// TwinCAT 3 PLC project PLC
// ProgramVersion: 3.1.4026.14
// libraries:
//   Tc2_Standard, * (Beckhoff Automation GmbH)
//   Tc2_System, * (Beckhoff Automation GmbH)
//   Tc2_Utilities, * (Beckhoff Automation GmbH)
//   Tc3_EventLogger, * (Beckhoff Automation GmbH)
//   Tc3_Module, * (Beckhoff Automation GmbH)
// project tree:
//   Devices/ Machine_Info.TcDUT, Pelletizer.TcDUT, VFD.TcDUT
//   FBs/ F_DPLC.TcPOU, Hour_Meter_FB.TcPOU, Send_Event_FB.TcPOU, SlaveStatus_FB.TcPOU
//   Global_Machine/ GVL_AirKnife.TcGVL, GVL_Pelletizer.TcGVL, GVL_System.TcGVL, GVL_Waterbath.TcGVL
//   / PlcTask.TcTTO
//   POUs/AirKnife/ Air_Knife_Control_Word.TcPOU, Check_Filter.TcPOU
//   POUs/ Main.TcPOU
//   POUs/Pelletizer/ DPLC.TcPOU, Machine_Limits.TcPOU, Pelletizer_Control.TcPOU, Pellet_Calibration.TcPOU
//   POUs/System/ Events.TcPOU, Imperial_Metric_Switching.TcPOU, Machine_Status.TcPOU, Scaling_And_Conversions.TcPOU, WritePersistentData_POU.TcPOU
//   POUs/WaterBath/ WaterBath_Control.TcPOU, Waterbath_Temp_Control.TcPOU
// real-time tasks:
//   TASK PlcTask: cycle T#10ms, priority 6, ADS port 350
// I/O:
//   DEVICE Device 1 (EtherCAT), AmsNetId 10.0.1.72.2.1
//     Rotor Drive [i550 Cabinet V06.04.xx]
//     Feedroll Drive [i550 Cabinet V06.04.xx]
// variable links:
//   PLC/PLC Instance <-> Device 1 (EtherCAT)/Feedroll Drive
//     PlcTask Inputs/GVL_Pelletizer.MyPelletizer.Feedroll_VFD.VFD_Actual_Current <-> TPDO (A) user config/Actual current
//     PlcTask Inputs/GVL_Pelletizer.MyPelletizer.Feedroll_VFD.VFD_Actual_Speed <-> TPDO (A) Velocity/Actual speed
//     PlcTask Inputs/GVL_Pelletizer.MyPelletizer.Feedroll_VFD.VFD_Actual_Torque <-> TPDO (A) user config/Actual torque
//     PlcTask Inputs/GVL_Pelletizer.MyPelletizer.Feedroll_VFD.VFD_Connection_Status <-> InfoData/State
//     PlcTask Inputs/GVL_Pelletizer.MyPelletizer.Feedroll_VFD.VFD_DC_Bus_Voltage <-> TPDO (A) user config/DC-bus voltage
//     PlcTask Inputs/GVL_Pelletizer.MyPelletizer.Feedroll_VFD.VFD_Digital_Input_Status <-> TPDO (A) user config/Digital input status
//     PlcTask Inputs/GVL_Pelletizer.MyPelletizer.Feedroll_VFD.VFD_Status_Word <-> TPDO (A) Velocity/CiA status word
//     PlcTask Outputs/GVL_Pelletizer.MyPelletizer.Feedroll_VFD.VFD_Control_Word <-> RPDO (A) Velocity/CiA control word
//     PlcTask Outputs/GVL_Pelletizer.MyPelletizer.Feedroll_VFD.VFD_Set_Speed <-> RPDO (A) Velocity/Set speed
//   PLC/PLC Instance <-> Device 1 (EtherCAT)/Rotor Drive
//     PlcTask Inputs/GVL_Pelletizer.MyPelletizer.Rotor_VFD.VFD_Actual_Current <-> TPDO (A) user config/Actual current
//     PlcTask Inputs/GVL_Pelletizer.MyPelletizer.Rotor_VFD.VFD_Actual_Speed <-> TPDO (A) Velocity/Actual speed
//     PlcTask Inputs/GVL_Pelletizer.MyPelletizer.Rotor_VFD.VFD_Actual_Torque <-> TPDO (A) user config/Actual torque
//     PlcTask Inputs/GVL_Pelletizer.MyPelletizer.Rotor_VFD.VFD_Connection_Status <-> InfoData/State
//     PlcTask Inputs/GVL_Pelletizer.MyPelletizer.Rotor_VFD.VFD_DC_Bus_Voltage <-> TPDO (A) user config/DC-bus voltage
//     PlcTask Inputs/GVL_Pelletizer.MyPelletizer.Rotor_VFD.VFD_Digital_Input_Status <-> TPDO (A) user config/Digital input status
//     PlcTask Inputs/GVL_Pelletizer.MyPelletizer.Rotor_VFD.VFD_Status_Word <-> TPDO (A) Velocity/CiA status word
//     PlcTask Outputs/GVL_Pelletizer.MyPelletizer.Rotor_VFD.VFD_Control_Word <-> RPDO (A) Velocity/CiA control word
//     PlcTask Outputs/GVL_Pelletizer.MyPelletizer.Rotor_VFD.VFD_Set_Speed <-> RPDO (A) Velocity/Set speed

CONFIGURATION PLC
    RESOURCE PLC ON TwinCAT3
        TASK PlcTask(INTERVAL := T#10ms, PRIORITY := 6);
        PROGRAM Main WITH PlcTask : Main;
        PROGRAM Air_Knife_Control_Word WITH PlcTask : Air_Knife_Control_Word;
        PROGRAM Machine_Status WITH PlcTask : Machine_Status;
        PROGRAM WaterBath_Control WITH PlcTask : WaterBath_Control;
        PROGRAM Pelletizer_Control WITH PlcTask : Pelletizer_Control;
        PROGRAM Events WITH PlcTask : Events;
        PROGRAM WritePersistentData_POU WITH PlcTask : WritePersistentData_POU;
    END_RESOURCE
END_CONFIGURATION

// ---- Devices/Machine_Info.TcDUT
TYPE Machine_Info :
STRUCT
	Machine_Serial_Number : STRING;
	Electrical_Bill_ID : STRING;
	Purchase_Order_Number : STRING;
	Work_Order_Number : STRING;
END_STRUCT
END_TYPE

// ---- Devices/Pelletizer.TcDUT
TYPE Pelletizer :
STRUCT
	Feedroll_VFD : VFD;
	Rotor_VFD : VFD;

	
	Feedroll_Driven_Pulley : REAL := 1;
	Feedroll_Drive_Pulley : REAL := 1;
	Feedroll_Diameter_Inch : REAL := 1.88;
	Feedroll_RPM: INT;
	Feedroll_Motor_RPM : INT;
	Feedroll_Feet_Per_Minute : REAL;
	Feedroll_Meters_Per_Minute : REAL;

	
	Rotor_Driven_Pulley : REAL := 1;
	Rotor_Drive_Pulley : REAL := 1;
	Rotor_Tooth_Count : REAL := 32;
	Rotor_RPM_Limit : REAL:= 1000;
	Rotor_RPM : REAL;
	Rotor_Motor_RPM : REAL;


	Pellet_Length_Inch_Input : REAL := 0.125;
	Pellet_Length_Calibration_Value : REAL := 1;
	Pellet_Length_Measured_Input : REAL;			//For use in Calibration
	
	
	Pelletizer_Info : Machine_Info;
	
	Pelletizer_Start : BOOL;
	Pelletizer_Fault : BOOL;
	Pelletizer_Fault_Reset : BOOL;
	Pelletizer_STO : BOOL;
END_STRUCT
END_TYPE

// ---- Devices/VFD.TcDUT
TYPE VFD :		//Map these directly to the Process Data.
STRUCT
	// PLC Inputs (Data read from the inverter) TPDOs
	VFD_Status_Word AT %I* : UINT;												//CiA Status Word
	VFD_Actual_Speed AT %I* : INT;												//VFD Actual Output RPM 
	VFD_Error_Code AT %I* : UINT;												//Error Message
	VFD_Actual_Torque AT %I* : INT;												//Instantaneous Torque of the Motor (In Percent x.x%)
	VFD_Actual_Current AT %I* : UINT;											//Instantaneous Current of the Motor (In Percent x.x%)
	VFD_DC_Bus_Voltage AT %I* : UDINT;											//Instantaneous DC Bus Voltage of the VFD (x.xxx Volts)
	VFD_Digital_Input_Status AT %I* : UDINT;

	VFD_Fault : BOOL;		 //:= VFD_Status_Word.3;				This callout doesnt seem to work during Runtime.						//This is part of the Status Word; Fault bit 3
	VFD_Connection_Status AT %I* : UINT;
	

	// PLC Outputs (Data written to the inverter) RPDOs
	VFD_Control_Word AT %Q* : UINT;												//State Machine for Controlling VFD (CiA)
	VFD_Set_Speed AT %Q* : INT;													//Sets the Speed of the VFD in RPM
	VFD_DigitalOutput1_Word AT %Q* : UINT;										//Map the NetInWord2 to something we can use.

	VFD_DigitalOutput1_Bit : BOOL := VFD_DigitalOutput1_Word.0;					//Break out just the bit that we use to control the digital output
	VFD_Fault_Reset : BOOL;	// := VFD_Control_Word.7;				This callout doesnt seem to work during Runtime.				//This is part of the Control Word; Fault Reset bit 7
	
END_STRUCT
END_TYPE

// ---- Global_Machine/GVL_AirKnife.TcGVL
{attribute 'qualified_only'}
VAR_GLOBAL PERSISTENT
	AirKnife_VFD : VFD;
	AirKnife_Start : BOOL;
	AirKnife_Percent_Speed_Input : REAL := 100;
	AirKnife_StartwithSystem : BOOL;
	AirKnife_StopwithSystem : BOOL;
	AirKnife_Analog_Input AT %I* : INT;
	AirKnife_Filter_Change_Setting : REAL := 15;
	AirKnife_Vacuum_Level : REAL;
END_VAR

// ---- Global_Machine/GVL_Pelletizer.TcGVL
{attribute 'qualified_only'}
///PERSISTENT VARIABLES: retain their value after an uncontrolled termination, a Reset cold or a new download of the PLC project. 
VAR_GLOBAL PERSISTENT	
//MyPelletizer structure. This is the main reference to all major variables for a pelletizer. 
// To call variables throughout program: Ex) GVL_Pelletizer.MyPelletizer.Feedroll_Motor.Motor_Rated_RPM := 1755;
	MyPelletizer : Pelletizer;
////////////////////////////////////////////////////////////////////////////////////////////////////
	

	Pellet_Length_Incorrect : BOOL;
END_VAR

// ---- Global_Machine/GVL_System.TcGVL
{attribute 'qualified_only'}
VAR_GLOBAL PERSISTENT
	
	RunTime : REAL;
	Emergency_Stop_Active : BOOL;
	Metric_Set_Bit : BOOL;

END_VAR

// ---- Global_Machine/GVL_Waterbath.TcGVL
{attribute 'qualified_only'}
VAR_GLOBAL PERSISTENT
	//OUTPUTS
	Prop_Valve AT %Q* : INT; 
	Pump_Start AT %Q* : BOOL;
	Pump_OL_Reset AT %Q* : BOOL;

	//INPUTS
	Process_Water_IN AT %I* : INT;
	Process_Water_OUT AT %I* : INT;
	Process_Water_FLOW AT %I* : INT;
	Pellet_Temp_Probe AT %I* : INT;
	Process_Water_Setpoint : INT;
	Waterbath_Connection_Status AT %I* : UINT;
	Waterbath_System_Control AT %I* : BOOL;
	Pump_Fault AT %I* : BOOL;

	
	//System Variables
	Waterbath_StartwithSystem : BOOL;
	Waterbath_StopwithSystem : BOOL;
	Waterbath_Start : BOOL;
	Waterbath_Running : BOOL;
	Waterbath_Local_Control : BOOL;
	
	//These are the HMI Variables after they are scaled correctly.
	Waterbath_SetPoint_Temp : LREAL;
	Waterbath_Actual_Temp : LREAL;
	Waterbath_Return_Temp : REAL;
	Waterbath_Flow_Rate : REAL;
	Waterbath_Pellet_Temperature : REAL;
	
	Waterbath_TempControl_Auto : BOOL;

	Waterbath_Delta_Temp : REAL;
	Waterbath_CalculatedBTULoss : REAL;
	
	Waterbath_Valve_Position_Percentage : REAL;
	
END_VAR

// ---- POUs/Main.TcPOU
PROGRAM Main
VAR PERSISTENT

	Hour_Meter : Hour_Meter_FB;

	connected : BOOL;
END_VAR

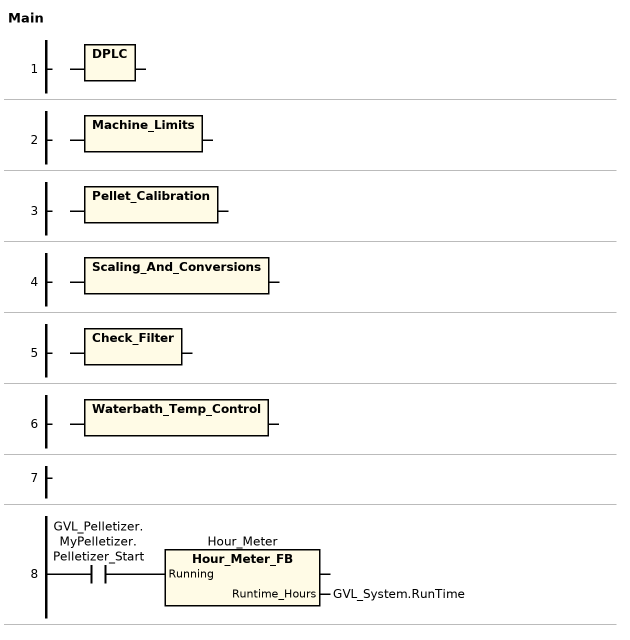
// NETWORK 1
DPLC();

// NETWORK 2
Machine_Limits();

// NETWORK 3
Pellet_Calibration();

// NETWORK 4
Scaling_And_Conversions();

// NETWORK 5
Check_Filter();

// NETWORK 6
Waterbath_Temp_Control();

// NETWORK 7

// NETWORK 8
Hour_Meter(Running := GVL_Pelletizer.MyPelletizer.Pelletizer_Start, Runtime_Hours => GVL_System.RunTime); // Hour_Meter_FB

END_PROGRAM

// ---- FBs/Hour_Meter_FB.TcPOU
FUNCTION_BLOCK Hour_Meter_FB
VAR_INPUT
	Running : BOOL;
END_VAR
VAR_OUTPUT
	Runtime_Hours : REAL;
END_VAR
VAR
	Running_Temp : BOOL;
	Minute_Timer : TON;
	Minutes : REAL;
	Hours : REAL;
	Elapsed : TIME;
END_VAR

Minute_Timer(IN:=Running_Temp , PT:=T#60S , Q=>, ET=>Elapsed );

IF Running THEN
	Running_Temp := TRUE;
END_IF
IF Minute_Timer.Q THEN
	Running_Temp := FALSE;
	Minutes := Minutes + 1;
END_IF
IF Minutes >= 60 THEN
	Minutes := 0;
	Hours := Hours + 1;
END_IF

Runtime_Hours := Hours;

END_FUNCTION_BLOCK

// ---- POUs/Pelletizer/DPLC.TcPOU
PROGRAM DPLC
VAR
	DPLC : F_DPLC;

	Calibrated_Pellet_Length : REAL;
END_VAR

GVL_Pelletizer.MyPelletizer.Feedroll_Motor_RPM := GVL_Pelletizer.MyPelletizer.Feedroll_VFD.VFD_Actual_Speed;

Calibrated_Pellet_Length := GVL_Pelletizer.MyPelletizer.Pellet_Length_Inch_Input * GVL_Pelletizer.MyPelletizer.Pellet_Length_Calibration_Value;

DPLC(
	Pellet_Length_Inch_Input		:= Calibrated_Pellet_Length,
	Feedroll_Diameter				:= GVL_Pelletizer.MyPelletizer.Feedroll_Diameter_Inch,
	Feedroll_Drive_Gear				:= GVL_Pelletizer.MyPelletizer.Feedroll_Drive_Pulley,
	Feedroll_Driven_Gear			:= GVL_Pelletizer.MyPelletizer.Feedroll_Driven_Pulley,
	Feedroll_Motor_RPM				:= GVL_Pelletizer.MyPelletizer.Feedroll_Motor_RPM,
	Rotor_Drive_Gear				:= GVL_Pelletizer.MyPelletizer.Rotor_Drive_Pulley,
	Rotor_Driven_Gear				:= GVL_Pelletizer.MyPelletizer.Rotor_Driven_Pulley,
	Rotor_Tooth_Count				:= GVL_Pelletizer.MyPelletizer.Rotor_Tooth_Count,
	Rotor_Motor_RPM					=> GVL_Pelletizer.MyPelletizer.Rotor_Motor_RPM,
	Rotor_RPM						=> GVL_Pelletizer.MyPelletizer.Rotor_RPM,
	Feedroll_Feet_Per_Minute		=> GVL_Pelletizer.MyPelletizer.Feedroll_Feet_Per_Minute
);
	
GVL_Pelletizer.MyPelletizer.Rotor_VFD.VFD_Set_Speed := REAL_TO_INT(GVL_Pelletizer.MyPelletizer.Rotor_Motor_RPM);


//Check for rotor speed exceeded. 
IF GVL_Pelletizer.MyPelletizer.Rotor_RPM >= GVL_Pelletizer.MyPelletizer.Rotor_RPM_Limit THEN
	GVL_Pelletizer.Pellet_Length_Incorrect := TRUE;
ELSE	
	GVL_Pelletizer.Pellet_Length_Incorrect := FALSE;
END_IF

END_PROGRAM

// ---- FBs/F_DPLC.TcPOU
FUNCTION_BLOCK F_DPLC
VAR_INPUT
	Pellet_Length_Inch_Input : REAL;
	
	//Feedroll
	Feedroll_Diameter : REAL;
	Feedroll_Drive_Gear : REAL;
	Feedroll_Driven_Gear : REAL;
	Feedroll_Motor_RPM : REAL;
	
	//Rotor
	Rotor_Drive_Gear : REAL;
	Rotor_Driven_Gear : REAL;
	Rotor_Tooth_Count : REAL;
	
END_VAR
VAR_OUTPUT
	
	Rotor_Motor_RPM : REAL;	//Commands the motor speed
	Rotor_RPM : REAL;		//Displays the actualy Rotor Speed
	
	Feedroll_Feet_Per_Minute : REAL;	//Displays the Actual Ft/min

END_VAR
VAR
	Feedroll_RPM : REAL;
	Feedroll_Inch_Per_Minute : REAL;

	Rotor_Cuts_Per_Minute : REAL;
END_VAR

Feedroll_RPM := Feedroll_Motor_RPM * (Feedroll_Drive_Gear / Feedroll_Driven_Gear);

Feedroll_Inch_Per_Minute := Feedroll_RPM * (Feedroll_Diameter * 3.14159);

Feedroll_Feet_Per_Minute := Feedroll_Inch_Per_Minute / 12.0;




Rotor_Cuts_Per_Minute := Feedroll_Inch_Per_Minute / Pellet_Length_Inch_Input;

Rotor_RPM := Rotor_Cuts_Per_Minute / Rotor_Tooth_Count;

Rotor_Motor_RPM := Rotor_RPM / (Rotor_Drive_Gear / Rotor_Driven_Gear);

END_FUNCTION_BLOCK

// ---- POUs/Pelletizer/Machine_Limits.TcPOU
PROGRAM Machine_Limits
VAR PERSISTENT
//For calculation purposes only. This calculates the min and max line speeds so that we can display these ranges on the speed gauges.

Feedroll_Motor_Rated_RPM : REAL := 1750;	
Feedroll_Motor_Rated_Hz : REAL := 60;		
Feedroll_Motor_Maximum_Hz : REAL;	
Feedroll_Motor_Minimum_Hz : REAL;	
Feedroll_Max_Ft_Per_Min : REAL;
Feedroll_Min_Ft_Per_Min  : REAL;
Feedroll_Motor_RPM_Per_Hz : REAL;
Feedroll_Pulley_Ratio : REAL;
Feedroll_Circumference_Feet : REAL := (GVL_Pelletizer.MyPelletizer.Feedroll_Diameter_Inch * 3.14159) / 12.0;

Rotor_Motor_Rated_RPM : REAL := 1750;	
Rotor_Motor_Rated_Hz : REAL := 60;	
Rotor_Motor_Maximum_Hz : REAL;	
Rotor_Motor_Minimum_Hz : REAL;	
Rotor_Max_RPM : REAL;
Rotor_Min_RPM : REAL;
Rotor_Motor_RPM_Per_Hz : REAL;
Rotor_Pulley_Ratio : REAL;


END_VAR

Feedroll_Pulley_Ratio := (GVL_Pelletizer.MyPelletizer.Feedroll_Drive_Pulley / GVL_Pelletizer.MyPelletizer.Feedroll_Driven_Pulley);

Feedroll_Motor_RPM_Per_Hz := Feedroll_Motor_Rated_RPM / Feedroll_Motor_Rated_Hz;

Feedroll_Max_Ft_Per_Min := ((Feedroll_Motor_RPM_Per_Hz * Feedroll_Motor_Maximum_Hz) * Feedroll_Pulley_Ratio) * Feedroll_Circumference_Feet;

Feedroll_Min_Ft_Per_Min := ((Feedroll_Motor_RPM_Per_Hz * Feedroll_Motor_Minimum_Hz) * Feedroll_Pulley_Ratio) * Feedroll_Circumference_Feet;



Rotor_Pulley_Ratio := (GVL_Pelletizer.MyPelletizer.Rotor_Drive_Pulley / GVL_Pelletizer.MyPelletizer.Rotor_Driven_Pulley);

Rotor_Motor_RPM_Per_Hz := Rotor_Motor_Rated_RPM / Rotor_Motor_Rated_Hz;

Rotor_Max_RPM := (Rotor_Motor_RPM_Per_Hz * Rotor_Motor_Maximum_Hz) * Rotor_Pulley_Ratio;

Rotor_Min_RPM := (Rotor_Motor_RPM_Per_Hz * Rotor_Motor_Minimum_Hz) * Rotor_Pulley_Ratio;

END_PROGRAM

// ---- POUs/Pelletizer/Pellet_Calibration.TcPOU
PROGRAM Pellet_Calibration
VAR
	SET_CALIBRATON_VALUE : BOOL;

	
	
	Pellet_Length_Temp_Cal_Val : REAL;
END_VAR

 Pellet_Length_Temp_Cal_Val :=  GVL_Pelletizer.MyPelletizer.Pellet_Length_Inch_Input / GVL_Pelletizer.MyPelletizer.Pellet_Length_Measured_Input;


IF SET_CALIBRATON_VALUE THEN
	GVL_Pelletizer.MyPelletizer.Pellet_Length_Calibration_Value := Pellet_Length_Temp_Cal_Val;
END_IF

END_PROGRAM

// ---- POUs/System/Scaling_And_Conversions.TcPOU
PROGRAM Scaling_And_Conversions
VAR
	Rotor_Actual_Torque_Scaled : REAL;
	Feedroll_Actual_Torque_Scaled : REAL;
	
	Rotor_Actual_Current_Scaled : REAL;
	Feedroll_Actual_Current_Scaled : REAL;
	AirKnife_Actual_Current_Scaled : REAL;
	
	Rotor_DC_Bus_Voltage_Scaled : REAL;
	Feedroll_DC_Bus_Voltage_Scaled : REAL;
	AirKnife_DC_Bus_Voltage_Scaled : REAL;
	

	AirKnife_Vacuum_Scaler : REAL := -4.0176; //-401.76 inH2O (-14.5PSI) / 100% = 4.0176
	
END_VAR

Rotor_Actual_Torque_Scaled := INT_TO_REAL(GVL_Pelletizer.MyPelletizer.Rotor_VFD.VFD_Actual_Torque) / 10;
Feedroll_Actual_Torque_Scaled := INT_TO_REAL(GVL_Pelletizer.MyPelletizer.Feedroll_VFD.VFD_Actual_Torque) / 10;

Rotor_Actual_Current_Scaled := UINT_TO_REAL(GVL_Pelletizer.MyPelletizer.Rotor_VFD.VFD_Actual_Current) / 10;
Feedroll_Actual_Current_Scaled := UINT_TO_REAL(GVL_Pelletizer.MyPelletizer.Feedroll_VFD.VFD_Actual_Current) / 10;
AirKnife_Actual_Current_Scaled := UINT_TO_REAL(GVL_Airknife.AirKnife_VFD.VFD_Actual_Current) / 10;


Rotor_DC_Bus_Voltage_Scaled := UDINT_TO_REAL(GVL_Pelletizer.MyPelletizer.Rotor_VFD.VFD_DC_Bus_Voltage) / 1000;
Feedroll_DC_Bus_Voltage_Scaled := UDINT_TO_REAL(GVL_Pelletizer.MyPelletizer.Feedroll_VFD.VFD_DC_Bus_Voltage) / 1000;
AirKnife_DC_Bus_Voltage_Scaled := UDINT_TO_REAL(GVL_AirKnife.AirKnife_Vfd.VFD_DC_Bus_Voltage) / 1000;

GVL_Airknife.AirKnife_Vacuum_Level := INT_TO_REAL(GVL_AirKnife.AirKnife_Analog_Input / 10) * AirKnife_Vacuum_Scaler;
//Sensor Scale:
//100% = -401.76 Inches of Water
//0% = 0 inches of water
//The analog input is read in as a percentage, not as 4-20ma

GVL_Waterbath.Waterbath_Actual_Temp := (((INT_TO_REAL(GVL_Waterbath.Process_Water_OUT) / 10) * 1.8) + 32.0);	//Convert thermocouple to Degrees F. 
GVL_Waterbath.Waterbath_Return_Temp := ((INT_TO_REAL(GVL_Waterbath.Process_Water_IN) / 30518.0) * 158);	//14F Degrees = 0 ADC; //158F Degrees = 30518
GVL_Waterbath.Waterbath_Pellet_Temperature := (((INT_TO_REAL(GVL_Waterbath.Pellet_Temp_Probe) / 10) * 1.8) + 32.0); //Convert thermocouple to Degrees F.

//0 - 198.129 GPM
GVL_Waterbath.Waterbath_Flow_Rate := ((INT_TO_REAL(GVL_WAterbath.Process_Water_FLOW) / 30518.0) * 198.129);

END_PROGRAM

// ---- POUs/AirKnife/Check_Filter.TcPOU
PROGRAM Check_Filter
VAR
	Change_Filter : BOOL;
	Startup_Timer : TON;
END_VAR

Startup_Timer(IN := GVL_airknife.AirKnife_Start,PT:=T#15S);	//Dont flag an alarm while it is starting up. Give it 15 seconds


IF (GVL_AirKnife.AirKnife_Filter_Change_Setting <= GVL_AirKnife.AirKnife_Vacuum_Level) AND (GVL_AirKnife.AirKnife_Vacuum_Level < -0.2) AND Startup_Timer.Q THEN
	Change_Filter := TRUE;
ELSE
	Change_Filter := FALSE;
END_IF

END_PROGRAM

// ---- POUs/WaterBath/Waterbath_Temp_Control.TcPOU
PROGRAM Waterbath_Temp_Control
VAR PERSISTENT
	Cooling_PID: FB_BasicPID;
	
	WaterbathPID_CycleTime : LREAL;
	Waterbath_ResetPID : BOOL;
	WaterbathPID_Kp : LREAL;
	WaterbathPID_Tn : LREAL;
	WaterbathPID_Tv : LREAL;
	WaterbathPID_Td : LREAL;
	
	WaterbathPID_ControlOutput : LREAL;
	WaterbathPID_ControlOutput_Temp : LREAL;

	WaterbathPID_ErrorStatus : UINT;
	
	
	
	
	//Erics Proportional Control
	
	Error : REAL;
	Gain : REAL;
	Deadband : REAL;
	
END_VAR

IF GVL_Waterbath.Waterbath_TempControl_Auto THEN
//	Cooling_PID(
//	fSetpointValue:= GVL_Waterbath.Waterbath_SetPoint_Temp, 
//	fActualValue:= GVL_Waterbath.Waterbath_Actual_Temp, 
//	bReset:= Waterbath_ResetPID, 
//	fCtrlCycleTime:= WaterbathPID_CycleTime, 
//	fKp:= WaterbathPID_Kp, 
//	fTn:= WaterbathPID_Tn, 
//	fTv:= WaterbathPID_Tv, 
//	fTd:= WaterbathPID_Td, 
//	fCtrlOutput=> WaterbathPID_ControlOutput, 
//	nErrorStatus=> WaterbathPID_ErrorStatus);


//Erics Proportional Algorithm
//Calculate error in temp difference
	Error := (GVL_Waterbath.Waterbath_Actual_Temp - GVL_Waterbath.Waterbath_SetPoint_Temp);	
//See if error is within deadband of 2 degrees
	IF ABS(Error) < Deadband THEN
		Error := 0;
	END_IF
//Error times the gain to set the output
	WaterbathPID_ControlOutput_Temp := Error * Gain;
//Limits on output. 	
	IF WaterbathPID_ControlOutput_Temp >= 100 THEN
		WaterbathPID_ControlOutput_Temp := 100;
	ELSIF WaterbathPID_ControlOutput_Temp < 0 THEN
		WaterbathPID_ControlOutput_Temp := 0;
	END_IF
	
	GVL_Waterbath.Waterbath_Valve_Position_Percentage := WaterbathPID_ControlOutput_Temp;
	WaterbathPID_ControlOutput := (GVL_Waterbath.Waterbath_Valve_Position_Percentage / 100) * 30518.0;
ELSE
	WaterbathPID_ControlOutput := (GVL_Waterbath.Waterbath_Valve_Position_Percentage / 100) * 30518.0;
END_IF

GVL_Waterbath.Prop_Valve := LREAL_TO_INT(WaterbathPID_ControlOutput);



GVL_Waterbath.Waterbath_Delta_Temp := GVL_Waterbath.Waterbath_Return_Temp - GVL_Waterbath.Waterbath_Actual_Temp;
GVL_Waterbath.Waterbath_CalculatedBTULoss := (GVL_Waterbath.Waterbath_Flow_Rate * (GVL_Waterbath.Waterbath_Delta_Temp) * 500.4);
// BTU Loss = Flow Rate In GPM (of water) x (Temperature Leaving Process - Temperature Entering Process) x 500.4

END_PROGRAM

// ---- POUs/AirKnife/Air_Knife_Control_Word.TcPOU
PROGRAM Air_Knife_Control_Word
VAR
	
	AirKnife_Lower_Status_Byte : UINT;
	
	Status_BitMask : UINT := 65280;

	
	Estop_Temp : bool;
END_VAR

GVL_AirKnife.AirKnife_VFD.VFD_Fault := GVL_AirKnife.AirKnife_VFD.VFD_Status_Word.3;	//Set fault bit equal to the status word fault bit.

IF GVL_AirKnife.AirKnife_VFD.VFD_Fault_Reset THEN
	//if the fault reset button was pressed, set the fault reset bit in the control word.
	GVL_AirKnife.AirKnife_VFD.VFD_Control_Word.7 := TRUE;
ELSE
	GVL_AirKnife.AirKnife_VFD.VFD_Control_Word.7 := FALSE;
END_IF



IF GVL_AirKnife.AirKnife_VFD.VFD_Fault THEN
	//If Faulted, then switch off drives
	GVL_AirKnife.AirKnife_VFD.VFD_Control_Word.0 := FALSE;
END_IF



IF GVL_Airknife.AirKnife_Stopwithsystem THEN
	Estop_Temp := GVL_Pelletizer.MyPelletizer.Pelletizer_STO;
ELSE
	Estop_Temp := TRUE;
END_IF

IF GVL_AirKnife.AirKnife_StartwithSystem THEN
	GVL_Airknife.AirKnife_Start := GVL_Pelletizer.MyPelletizer.Pelletizer_Start;
END_IF


	//If the Start button on the HMI is pressed, OR it is set to start with the rest of the system. The checkbox must be set and pelletizer must be started.
IF GVL_AirKnife.AirKnife_Start AND Estop_Temp THEN
	
//Feedroll Case Statement
	AirKnife_Lower_Status_Byte := GVL_AirKnife.AirKnife_VFD.VFD_Status_Word OR Status_BitMask;	// Bitwise OR with bits 7-15 of status word because we dont care about them for control.
	
	CASE AirKnife_Lower_Status_Byte OF
		65392: //Voltage Enabled, Switch On Disabled.
		GVL_AirKnife.AirKnife_VFD.VFD_Control_Word := 6;	//Enable Voltage, Disable Quick Stop	
	
		65360: //Voltage Enabled, Switch On Disabled.
		GVL_AirKnife.AirKnife_VFD.VFD_Control_Word := 6;	//Enable Voltage, Disable Quick Stop
	
		65329: //Ready To Switch On, Voltage Enabled, Quick Stop Disabled.
		GVL_AirKnife.AirKnife_VFD.VFD_Control_Word := 7;	//Enable Voltage, Disable Quick Stop, Switch On
	
		65331: //Ready To Switch On, Switched On, Voltage Enabled, Quick Stop Disabled.
		GVL_AirKnife.AirKnife_VFD.VFD_Control_Word := 15;	//Enable Voltage, Disable Quick Stop, Switch On, Enable Operation
	
		65335: //Ready To Switch On, Switched On, Operation Enabled, Voltage Enabled, Quick Stop Disabled.
		GVL_AirKnife.AirKnife_VFD.VFD_Control_Word.0 := TRUE;	//Switch On Bit. 
	END_CASE;

ELSE	
	//If we are not running, switch off Drives
	GVL_AirKnife.AirKnife_VFD.VFD_Control_Word.0 := 0;
END_IF



//The last thing is to scale the motor RPM to a percentage.
GVL_AirKnife.AirKnife_VFD.VFD_Set_Speed := REAL_TO_INT((3450 / 100) * GVL_AirKnife.AirKnife_Percent_Speed_Input);
// I should add some parameters for the air knife settings screen to the max RPM

END_PROGRAM

// ---- POUs/System/Machine_Status.TcPOU
PROGRAM Machine_Status
VAR
	AirKnife_Status_String : STRING;
	AirKnife_Disconnected : BOOL;
	AirKnife_Connected : bool;
	
	Rotor_Status_String : STRING;
	Rotor_Disconnected : BOOL;
	
	Feedroll_Status_String : STRING;
	Feedroll_Disconnected : BOOL;
	
	Pelletizer_Status_String : STRING;
	
	Waterbath_Status_String : STRING;
	Waterbath_Disconnected : BOOL;
	Waterbath_Connected : BOOL;
	
END_VAR


Rotor_Status_String := SlaveStatus_FB(GVL_Pelletizer.MyPelletizer.Rotor_VFD.VFD_Connection_Status, Slave_Disconnected => Rotor_Disconnected);
Feedroll_Status_String := SlaveStatus_FB(GVL_Pelletizer.MyPelletizer.Feedroll_VFD.VFD_Connection_Status, Slave_Disconnected => Feedroll_Disconnected);

IF Rotor_Disconnected OR Feedroll_Disconnected THEN
	Pelletizer_Status_String := CONCAT(Rotor_Status_String, Feedroll_Status_String);
ELSE
	Pelletizer_Status_String := 'Slave in OP state';
END_IF


AirKnife_Status_String := SlaveStatus_FB(GVL_AirKnife.AirKnife_VFD.VFD_Connection_Status, Slave_Disconnected => AirKnife_Disconnected);
AirKnife_connected := NOT Airknife_Disconnected;

Waterbath_Status_String := SlaveStatus_FB(GVL_Waterbath.Waterbath_Connection_Status, Slave_Disconnected => Waterbath_Disconnected);
Waterbath_Connected := NOT Waterbath_Disconnected;

END_PROGRAM

// ---- FBs/SlaveStatus_FB.TcPOU
FUNCTION SlaveStatus_FB : STRING
VAR_INPUT
	InfoData_State : UINT; // Input variable containing the status bitmask
END_VAR
VAR
	Bit8_Message : STRING;
	Bitmask : UINT := 16#FFF0;
	Masked_State: UINT;
END_VAR
VAR_OUTPUT
	Slave_Disconnected : BOOL;
END_VAR

Masked_State := bitmask OR InfoData_State;


IF InfoData_State.8 THEN
	Bit8_Message := ' - Slave NOT present ';
	Slave_Disconnected := TRUE;
ELSE
	Bit8_Message := '';
	Slave_Disconnected := FALSE;
END_IF
	



CASE Masked_State OF
    16#FFF1: SlaveStatus_FB 		:= 'Slave in INIT state';		//16#___1; // Slave in 'INIT' state
    16#FFF2: SlaveStatus_FB 		:= 'Slave in PREOP state';		//16#___2; // Slave in 'PREOP' state
    16#FFF3: SlaveStatus_FB 		:= 'Slave in BOOT state';		//16#___3; // Slave in 'BOOT' state
    16#FFF4: SlaveStatus_FB 		:= 'Slave in SAFEOP state';		//16#___4; // Slave in 'SAFEOP' state
    16#FFF8: SlaveStatus_FB 		:= 'Slave in OP state';			//16#___8 Slave in 'OP' state
ELSE
    // Handle invalid input or unknown status
    SlaveStatus_FB := 'Abnormal Status'; // Set an appropriate error value
	Slave_Disconnected := TRUE;
END_CASE;

SlaveStatus_FB := CONCAT(SlaveStatus_FB, Bit8_message);	//Add both messages to display.



//Breakdown of Statuses for Infomation, we dont care about all of them. Just the EtherCAT State and the slave Not present bit. 
//0x___1 = Slave in 'INIT' state
//0x___2 = Slave in 'PREOP' state
//0x___3 = Slave in 'BOOT' state
//0x___4 = Slave in 'SAFEOP' state
//0x___8 = Slave in 'OP' state
//0x001_ = Slave signals error
//0x002_ = Invalid vendorId, productCode... read
//0x004_ = Initialization error occurred
//0x008_ = Slave disabled
//0x010_ = Slave not present
//0x020_ = Slave signals link error
//0x040_ = Slave signals missing link
//0x080_ = Slave signals unexpected link
//0x100_ = Communication port A
//0x200_ = Communication port B
//0x400_ = Communication port C
//0x800_ = Communication port D

END_FUNCTION

// ---- POUs/WaterBath/WaterBath_Control.TcPOU
PROGRAM WaterBath_Control
VAR
	
	Estop_Temp : bool;

END_VAR

IF GVL_Waterbath.Waterbath_StopwithSystem THEN		//if the pelletizer estop is pressed AND the setting for system stop is set, then stop with an estop.
	Estop_Temp := GVL_Pelletizer.MyPelletizer.Pelletizer_STO;
ELSE
	Estop_Temp := TRUE;
END_IF




IF GVL_Waterbath.Waterbath_StartwithSystem THEN
	GVL_Waterbath.Waterbath_Start := GVL_Pelletizer.MyPelletizer.Pelletizer_Start;
END_IF




IF GVL_Waterbath.Waterbath_Start AND Estop_Temp THEN
	GVL_Waterbath.Pump_Start := TRUE;
ELSE
	GVL_Waterbath.Pump_Start := FALSE;
END_IF


GVL_Waterbath.Waterbath_Local_Control := NOT GVL_Waterbath.Waterbath_System_Control;

END_PROGRAM

// ---- POUs/Pelletizer/Pelletizer_Control.TcPOU
PROGRAM Pelletizer_Control
VAR
	Pelletizer_Lower_Status_Byte : UINT;
	
	Status_BitMask : UINT := 65280;
	DigitalInputStatus: INT;
	


END_VAR

//Bit 15 is digital input 1 which is the pelletizer control relay. If both of these are ON, we are in a started state.
IF (GVL_Pelletizer.MyPelletizer.Feedroll_VFD.VFD_Digital_Input_Status.16 = TRUE) AND (GVL_Pelletizer.MyPelletizer.Rotor_VFD.VFD_Digital_Input_Status.16 = TRUE) THEN
	GVL_Pelletizer.MyPelletizer.Pelletizer_Start := TRUE;
ELSE	
	GVL_Pelletizer.MyPelletizer.Pelletizer_Start := FALSE;
END_IF




//Fault Handling
GVL_Pelletizer.MyPelletizer.Feedroll_VFD.VFD_Fault := GVL_Pelletizer.MyPelletizer.Feedroll_VFD.VFD_Status_Word.3;
GVL_Pelletizer.MyPelletizer.Rotor_VFD.VFD_Fault := GVL_Pelletizer.MyPelletizer.Rotor_VFD.VFD_Status_Word.3;
//Overall Machine Fault if one or both drives faulted. 
IF (GVL_Pelletizer.MyPelletizer.Feedroll_VFD.VFD_Fault) OR (GVL_Pelletizer.MyPelletizer.Rotor_VFD.VFD_Fault) THEN
	GVL_Pelletizer.MyPelletizer.Pelletizer_Fault := TRUE;
ELSE
	GVL_Pelletizer.MyPelletizer.Pelletizer_Fault := FALSE;	
END_IF



//Reset faults
IF GVL_Pelletizer.MyPelletizer.Pelletizer_Fault_Reset THEN
	GVL_Pelletizer.MyPelletizer.Feedroll_VFD.VFD_Fault_Reset := TRUE;
	GVL_Pelletizer.MyPelletizer.Rotor_VFD.VFD_Fault_Reset := TRUE;
ELSE
	GVL_Pelletizer.MyPelletizer.Feedroll_VFD.VFD_Fault_Reset := FALSE;
	GVL_Pelletizer.MyPelletizer.Rotor_VFD.VFD_Fault_Reset := FALSE;
END_IF
//Set Reset
GVL_Pelletizer.MyPelletizer.Feedroll_VFD.VFD_Control_Word.7 := GVL_Pelletizer.MyPelletizer.Feedroll_VFD.VFD_Fault_reset;
GVL_Pelletizer.MyPelletizer.Rotor_VFD.VFD_Control_Word.7 := GVL_Pelletizer.MyPelletizer.Rotor_VFD.VFD_Fault_Reset;

GVL_Pelletizer.MyPelletizer.Pelletizer_STO := GVL_Pelletizer.MyPelletizer.Feedroll_VFD.VFD_Status_Word.15 OR GVL_Pelletizer.MyPelletizer.rotor_VFD.VFD_Status_Word.15;

END_PROGRAM

// ---- POUs/System/Events.TcPOU
PROGRAM Events
VAR
	Send_Start_Event : Send_Event_FB;
	Start_Event  : TcEventEntry := TC_Events.Pelletizer_Events.Start_Button_Event;
	
	Send_Stop_Event : Send_Event_FB;
	Stop_Event  : TcEventEntry := TC_Events.Pelletizer_Events.Stop_Button_Event;
//////////////////////////////////////////////////////////////////////////////////////////////////////////////////
	Send_EmergencyStop_Event : Send_Event_FB;
	EmergencyStop_Event : TcEventEntry := TC_Events.Pelletizer_Events.Emergency_Stop_Set_Event;

	Send_EmergencyStop_Reset_Event : Send_Event_FB;
	EmergencyStop_Reset_Event : TcEventEntry := TC_Events.Pelletizer_Events.Emergency_Stop_Reset_Event;
//////////////////////////////////////////////////////////////////////////////////////////////////////////////////	
	Send_Feedroll_Drive_Fault_Event : Send_Event_FB;
	Feedroll_Drive_Fault_Event : TcEventEntry := TC_Events.Pelletizer_Events.Feedroll_Drive_Fault_Event;
	
	Send_Feedroll_Drive_Fault_Reset_Event : Send_Event_FB;
	Feedroll_Drive_Fault_Reset_Event : TcEventEntry := TC_Events.Pelletizer_Events.Feedroll_Drive_Fault_Reset_Event;
//////////////////////////////////////////////////////////////////////////////////////////////////////////////////	
	Send_Rotor_Drive_Fault_Event : Send_Event_FB;
	Rotor_Drive_Fault_Event : TcEventEntry := TC_Events.Pelletizer_Events.Rotor_Drive_Fault_Event;
	
	Send_Rotor_Drive_Fault_Reset_Event : Send_Event_FB;
	Rotor_Drive_Fault_Reset_Event : TcEventEntry := TC_Events.Pelletizer_Events.Rotor_Drive_Fault_Reset_Event;
//////////////////////////////////////////////////////////////////////////////////////////////////////////////////
	Send_Machine_Shutdown_Event : Send_Event_FB;
	Machine_Shutdown_Event : TcEventEntry := TC_Events.Pelletizer_Events.Machine_Shutdown_Event;	
	
	Send_Machine_PowerOn_Event : Send_Event_FB;
	Machine_PowerOn_Event : TcEventEntry := TC_Events.Pelletizer_Events.Machine_PowerOn_Event;
//////////////////////////////////////////////////////////////////////////////////////////////////////////////////	
	Send_Exceeded_Pellet_Length_Event : Send_Event_FB;
	Exceeded_Pellet_Length_Event : TcEventEntry := TC_Events.Pelletizer_Events.PelletLength_Exceeded_Event;	
//////////////////////////////////////////////////////////////////////////////////////////////////////////////////	
	Send_Change_Filter_Event : Send_Event_FB;
	Change_Filter_Event : TcEventEntry := TC_Events.AirKnife_Events.Change_Filter_Event;	
	
	Send_Filter_OKAY_Event : Send_Event_FB;
	Filter_OKAY_Event : TcEventEntry := TC_Events.AirKnife_Events.Filter_OKAY_Event;
//////////////////////////////////////////////////////////////////////////////////////////////////////////////////	
	Send_Local_Mode_Active : Send_Event_FB;
	Local_Mode_Active : TcEventEntry := TC_Events.Waterbath_Events.Local_Mode_Active;
	
	Send_Remote_Mode_Active : Send_Event_FB;
	Remote_Mode_Active : TcEventEntry := TC_Events.Waterbath_Events.Remote_Mode_Active;
//////////////////////////////////////////////////////////////////////////////////////////////////////////////////	
	Send_Pump_Start_Event : Send_Event_FB;
	Pump_Start_Event : TcEventEntry := TC_Events.Waterbath_Events.Pump_Start_Event;
	
	Send_Pump_Stop_Event : Send_Event_FB;
	Pump_Stop_Event : TcEventEntry := TC_Events.Waterbath_Events.Pump_Stop_Event;
//////////////////////////////////////////////////////////////////////////////////////////////////////////////////	
	
	First_Scan : BOOL := False;	
END_VAR

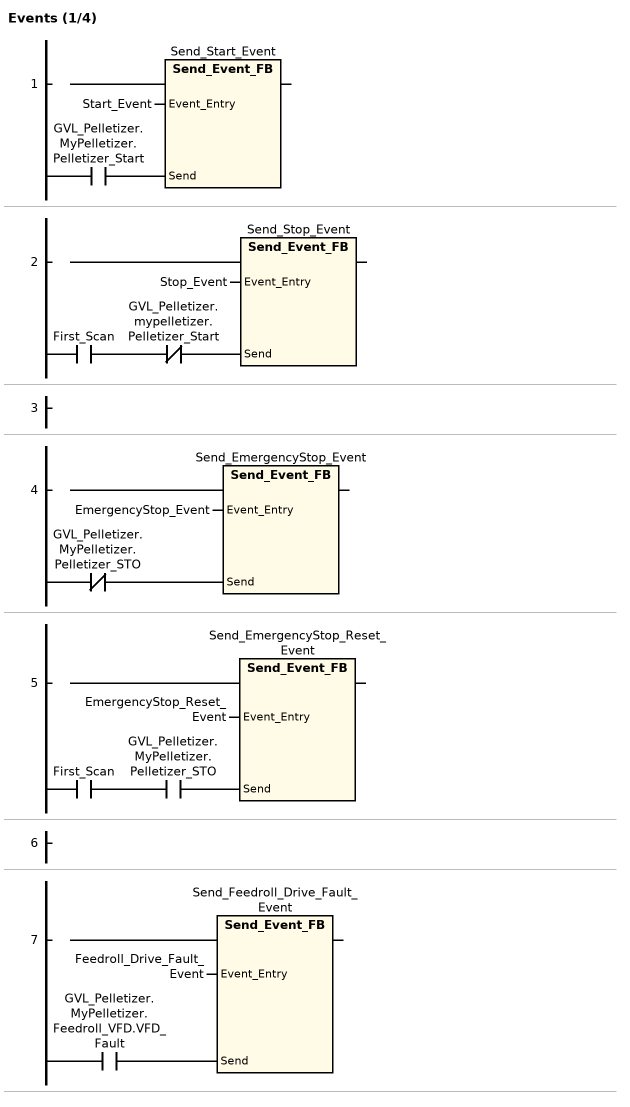
// NETWORK 1
Send_Start_Event(Event_Entry := Start_Event, Send := GVL_Pelletizer.MyPelletizer.Pelletizer_Start); // Send_Event_FB

// NETWORK 2
Send_Stop_Event(Event_Entry := Stop_Event, Send := First_Scan AND NOT GVL_Pelletizer.mypelletizer.Pelletizer_Start); // Send_Event_FB

// NETWORK 3

// NETWORK 4
Send_EmergencyStop_Event(Event_Entry := EmergencyStop_Event, Send := NOT GVL_Pelletizer.MyPelletizer.Pelletizer_STO); // Send_Event_FB

// NETWORK 5
Send_EmergencyStop_Reset_Event(Event_Entry := EmergencyStop_Reset_Event, Send := First_Scan AND GVL_Pelletizer.MyPelletizer.Pelletizer_STO); // Send_Event_FB

// NETWORK 6

// NETWORK 7
Send_Feedroll_Drive_Fault_Event(Event_Entry := Feedroll_Drive_Fault_Event, Send := GVL_Pelletizer.MyPelletizer.Feedroll_VFD.VFD_Fault); // Send_Event_FB

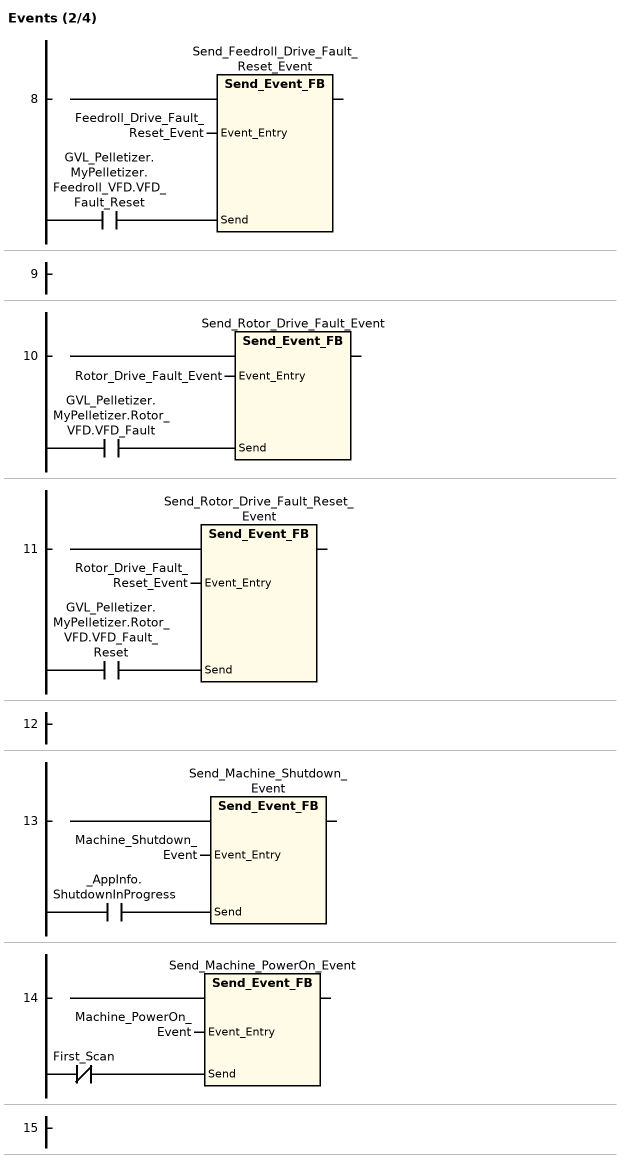
// NETWORK 8
Send_Feedroll_Drive_Fault_Reset_Event(Event_Entry := Feedroll_Drive_Fault_Reset_Event, Send := GVL_Pelletizer.MyPelletizer.Feedroll_VFD.VFD_Fault_Reset); // Send_Event_FB

// NETWORK 9

// NETWORK 10
Send_Rotor_Drive_Fault_Event(Event_Entry := Rotor_Drive_Fault_Event, Send := GVL_Pelletizer.MyPelletizer.Rotor_VFD.VFD_Fault); // Send_Event_FB

// NETWORK 11
Send_Rotor_Drive_Fault_Reset_Event(Event_Entry := Rotor_Drive_Fault_Reset_Event, Send := GVL_Pelletizer.MyPelletizer.Rotor_VFD.VFD_Fault_Reset); // Send_Event_FB

// NETWORK 12

// NETWORK 13
Send_Machine_Shutdown_Event(Event_Entry := Machine_Shutdown_Event, Send := _AppInfo.ShutdownInProgress); // Send_Event_FB

// NETWORK 14
Send_Machine_PowerOn_Event(Event_Entry := Machine_PowerOn_Event, Send := NOT First_Scan); // Send_Event_FB

// NETWORK 15

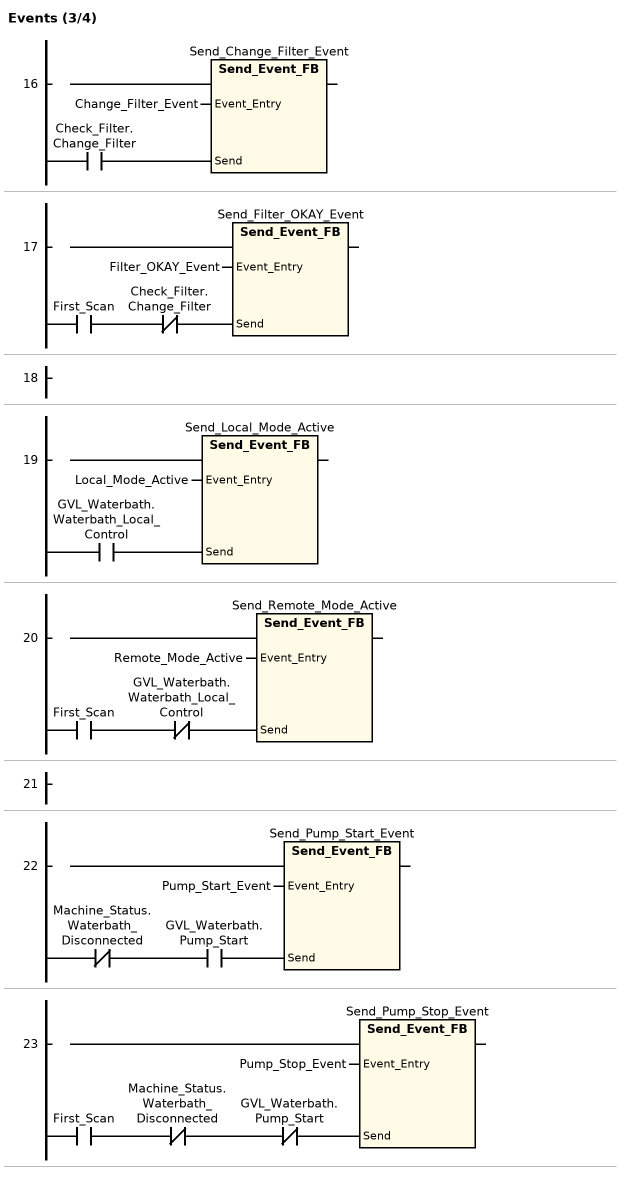
// NETWORK 16
Send_Change_Filter_Event(Event_Entry := Change_Filter_Event, Send := Check_Filter.Change_Filter); // Send_Event_FB

// NETWORK 17
Send_Filter_OKAY_Event(Event_Entry := Filter_OKAY_Event, Send := First_Scan AND NOT Check_Filter.Change_Filter); // Send_Event_FB

// NETWORK 18

// NETWORK 19
Send_Local_Mode_Active(Event_Entry := Local_Mode_Active, Send := GVL_Waterbath.Waterbath_Local_Control); // Send_Event_FB

// NETWORK 20
Send_Remote_Mode_Active(Event_Entry := Remote_Mode_Active, Send := First_Scan AND NOT GVL_Waterbath.Waterbath_Local_Control); // Send_Event_FB

// NETWORK 21

// NETWORK 22
Send_Pump_Start_Event(Event_Entry := Pump_Start_Event, Send := NOT Machine_Status.Waterbath_Disconnected AND GVL_Waterbath.Pump_Start); // Send_Event_FB

// NETWORK 23
Send_Pump_Stop_Event(Event_Entry := Pump_Stop_Event, Send := First_Scan AND NOT Machine_Status.Waterbath_Disconnected AND NOT GVL_Waterbath.Pump_Start); // Send_Event_FB

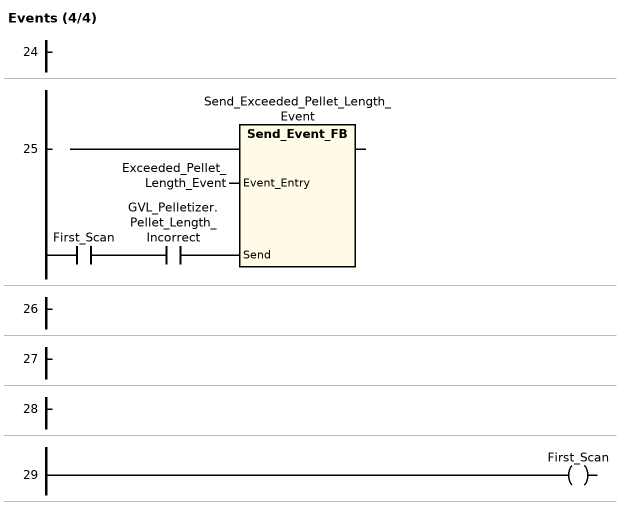
// NETWORK 24

// NETWORK 25
Send_Exceeded_Pellet_Length_Event(Event_Entry := Exceeded_Pellet_Length_Event, Send := First_Scan AND GVL_Pelletizer.Pellet_Length_Incorrect); // Send_Event_FB

// NETWORK 26

// NETWORK 27

// NETWORK 28

// NETWORK 29
First_Scan := TRUE;

END_PROGRAM

// ---- FBs/Send_Event_FB.TcPOU
FUNCTION_BLOCK Send_Event_FB
VAR_INPUT
	Event_Entry : TcEventEntry;
	Send : BOOL;

END_VAR
VAR
	fbMessage : FB_TcMessage;
	Trigger : R_TRIG;
END_VAR

Trigger(CLK:=Send);


IF Trigger.Q THEN
	fbMessage.CreateEx(Event_Entry, 0);
    fbMessage.Send(0);
	fbMessage.Release();
END_IF




// You must create the Event using CreateEx. The input to this is the exact Event Entry you want to send.
//Call this function and enable it by turning on the SEND input. This will send one message when the input is True. 
//In order to send subsequent messages, the input must go from False back to True.


// Event Entry:
// Example Callout: TC_Events.Pelletizer_Events.Start_Button_Event
// The Event list is under Type System, Click "Event Classes" tab on right side.
// "Pelletizer Events" should be one of the last items on the list
// Right Click > Edit


//An idea would to create a structure/enumeration of these events to call them by number. 
//I have not done this yet.

END_FUNCTION_BLOCK

// ---- POUs/System/WritePersistentData_POU.TcPOU
PROGRAM WritePersistentData_POU
VAR
    NETID  : T_AmsNetId := '';		//AMS Net ID. An empty string designates the local machine.
    PORT   : UINT := 851;			//Always port 851 for our simple stuff
    START  : BOOL;					//Start bit
    TMOUT  : TIME := DEFAULT_ADS_TIMEOUT;	
    fbWritePersistentData : FB_WritePersistentData;		//Instance name
    fbR_Trig              : R_TRIG;						//Use a rising edge trigger. This coupled with a pelletizer Running command gives us deterministic saving of variables.
END_VAR



// This POU is only used on PCs without integrated UPS Backup. 
// All Beckhoff controllers have this function integrated.
// This was written in for the PH25-Beta machine which used a Teguar 3rd party PC as its contoller.
//You can delete this whole POU if you are using a Beckhoff controller.




fbR_Trig( CLK:=GVL_Pelletizer.MyPelletizer.Pelletizer_Start);
IF fbR_Trig.Q THEN
	fbWritePersistentData(NETID:=NETID,PORT:=PORT, START := GVL_Pelletizer.MyPelletizer.Pelletizer_Start, TMOUT:=TMOUT, MODE:=1);
ELSE
    fbWritePersistentData( START:=FALSE);
END_IF

END_PROGRAM

// ---- POUs/System/Imperial_Metric_Switching.TcPOU
PROGRAM Imperial_Metric_Switching
VAR PERSISTENT
	Pellet_Length_Displayed : REAL;
	Pellet_Length_Metric_Input : REAL;
	//Pellet_Length_Imperial_Input : REAL;	Uses GVL_Pelletizer.Pellet_Length_Inch_Input
	
	Line_Speed_Displayed : REAL;
	Line_Speed_Metric_Input : REAL;
	//FeedRate_Feet_Per_Minute_Input : REAL; Uses GVL_Pelletizer.Feedroll
	

END_VAR

IF GVL_System.Metric_Set_Bit THEN		//Convert to Metric

	// Converts the displayed input value into Imperial Inches for the PLCs calculations. The Metric numbers are for display only.
	Pellet_Length_Displayed := Pellet_Length_Metric_Input;
	GVL_Pelletizer.MyPelletizer.Pellet_Length_Inch_Input := Pellet_Length_Metric_Input / 25.4;
		
	// Converts the displayed input speed into Imperial feet per minute for the PLCs calculations. The Metric numbers are for display only.	
	// This also converts the internal calculations back into Metric for viewing.
	//Line_Speed_Displayed := Line_Speed_Metric_Input;
	//GVL_Feedroll.FeedRate_Feet_Per_Minute_Input := Line_Speed_Metric_Input / 0.30480;
ELSE		//Stay in Imperial

	Pellet_Length_Displayed := GVL_Pelletizer.MyPelletizer.Pellet_Length_Inch_Input;
	Pellet_Length_Metric_Input := GVL_Pelletizer.MyPelletizer.Pellet_Length_Inch_Input * 25.4;
		
	//Line_Speed_Displayed := GVL_Feedroll.FeedRate_Feet_Per_Minute_Input;
	//Line_Speed_Metric_Input := GVL_Feedroll.FeedRate_Feet_Per_Minute_Input * 0.30480;
END_IF

END_PROGRAM
